// TIA Portal V20 export
DATA_BLOCK "zPMC_Map_DB_04"   // DB398
// stored: InstanceOfName CITI_Logic.zPMC_Map, InstanceOfType FB, Namespace Citi_logic
"CITI_Logic.zPMC_Map"
   // VAR_INPUT
   //    IN_AssistanceCall : Array[1..8] of Bool;
   //    IN_AssistanceCallAck : Array[1..8] of Bool;
   //    IN_Configuration : "CITI_Logic.zp_CITI_Configuration";
   //    IN_Data : "CITI_Logic.PMC_Input_Data";
   // END_VAR
   // VAR_OUTPUT
   //    OUT_Flasher_1Hz : Bool;
   //    OUT_Team_Leader_Call_Out : Bool;
   //    OUT_ShiftNumber : Byte;
   // END_VAR
   // VAR_IN_OUT
   //    PMC_Data : "CITI_Logic.zp_CITIData";
   // END_VAR
   // VAR
   //    MM_FaultWord_Zero : Bool;
   //    CycleTime_RUNNING_FB : Bool;
   //    Cycle_END_OneShot_FB : Bool;
   //    System_Time_Tick : Time;
   //    Present_Time_Tick : Int;
   //    Previous_Time_Tick : Int;
   //    Difference_Time_Tick : Int;
   //    Difference_Time_DInt : DInt;
   //    CurrentProcessTime_DInt : DInt;
   //    CurrentPTimeConvertDInt : DInt;
   //    CurrentHeartBeatTim_DInt : DInt;
   //    ShiftResetHold : Bool;
   //    HeartBeatSetOneShot : Bool;
   //    DataReadySetup : Bool;
   //    CurrentLoadTime_DInt : DInt;
   //    CurrentLTimeConvertDInt : DInt;
   //    CurrentUnLoadTime_DInt : DInt;
   //    CurrentUTimeConvertDInt : DInt;
   //    CurrentPUNRdyDly_DInt : DInt;
   //    TimerForDataReadySetup : DInt;
   //    TimerForCycleTimeReady : DInt;
   //    TimerForFaultDelay : DInt;
   //    Last_PUN_Data : String[20];
   //    FTQ_CurrDataRdyTime_DInt : DInt;
   //    FTQ_Internal_Data_Ready : Bool;
   //    NullChar : Char;
   //    OneShotFirstScan : Bool;
   //    PUN_Is_NOT_Equal : Bool;
   //    PartType_NOT_Unknown : Bool;
   //    PartType_NOT_Equal : Bool;
   //    FaultStringIs9902 : Bool;
   //    TimerForFlasher : DInt;
   //    FB_OneShot : Array[1..32] of Bool;
   //    CurDTL { ExternalAccessible := 'False'; ExternalVisible := 'False'; ExternalWritable := 'False'} : DTL;
   //    ON { ExternalAccessible := 'False'; ExternalVisible := 'False'; ExternalWritable := 'False'} : Bool;
   //    OFF { ExternalAccessible := 'False'; ExternalVisible := 'False'; ExternalWritable := 'False'} : Bool;
   //    Temp_DINT { ExternalAccessible := 'False'; ExternalVisible := 'False'; ExternalWritable := 'False'} : DInt;
   //    Temp_INT { ExternalAccessible := 'False'; ExternalVisible := 'False'; ExternalWritable := 'False'} : Int;
   //    Temp_LastCycle_Time { ExternalAccessible := 'False'; ExternalVisible := 'False'; ExternalWritable := 'False'} : DInt;
   //    FTQ_t_ZERO { ExternalAccessible := 'False'; ExternalVisible := 'False'; ExternalWritable := 'False'} : Int;
   //    Fault_Load_Delay_Other_or_Unknown : IEC_TIMER;
   //    FlasherRatex2 { S7_SetPoint := 'True'} : DInt;
   // END_VAR
BEGIN
END_DATA_BLOCK
